FUNCTION_BLOCK CRANE_1_PUBLISH (* Composite Function Block Type *)
  (* Standard: 61499-2 *)
  (* Version 1.0, 2019-04-13, adeel *)
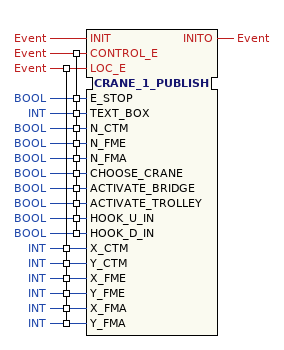
  EVENT_INPUT
    INIT; (* Initialization Request *)
    CONTROL_E WITH E_STOP, TEXT_BOX, N_CTM, N_FME, N_FMA, CHOOSE_CRANE, ACTIVATE_BRIDGE, ACTIVATE_TROLLEY, HOOK_U_IN, HOOK_D_IN; (* Normal Execution Request *)
    LOC_E WITH X_CTM, Y_CTM, X_FME, Y_FME, X_FMA, Y_FMA;
  END_EVENT
  EVENT_OUTPUT
    INITO; (* Initialization Confirm *)
  END_EVENT
  VAR_INPUT
    E_STOP : BOOL;
    TEXT_BOX : INT;
    N_CTM : BOOL;
    N_FME : BOOL;
    N_FMA : BOOL;
    CHOOSE_CRANE : BOOL;
    ACTIVATE_BRIDGE : BOOL;
    ACTIVATE_TROLLEY : BOOL;
    HOOK_U_IN : BOOL;
    HOOK_D_IN : BOOL;
    X_CTM : INT;
    Y_CTM : INT;
    X_FME : INT;
    Y_FME : INT;
    X_FMA : INT;
    Y_FMA : INT;
  END_VAR
  FBS
    PUBLISH_1 : PUBLISH_1(QI := 1, ID := opc_ua[opc.tcp://%CRANE1_IP%:4840#/Objects/1:CRANE1C/N_CTM/IN]);
    PUBLISH_1_1 : PUBLISH_1(QI := 1, ID := opc_ua[opc.tcp://%CRANE1_IP%:4840#/Objects/1:CRANE1B/TEXT_BOX/IN]);
    PUBLISH_1_2 : PUBLISH_1(QI := 1, ID := opc_ua[opc.tcp://%CRANE1_IP%:4840#/Objects/1:CRANE1K/X_CTM/IN]);
    PUBLISH_1_3 : PUBLISH_1(QI := 1, ID := opc_ua[opc.tcp://%CRANE1_IP%:4840#/Objects/1:CRANE1A/E_STOP/IN]);
    PUBLISH_1_4 : PUBLISH_1(QI := 1, ID := opc_ua[opc.tcp://%CRANE1_IP%:4840#/Objects/1:CRANE1L/Y_CTM/IN]);
    PUBLISH_1_5 : PUBLISH_1(QI := 1, ID := opc_ua[opc.tcp://%CRANE1_IP%:4840#/Objects/1D:CRANE1/N_FME/IN]);
    PUBLISH_1_6 : PUBLISH_1(QI := 1, ID := opc_ua[opc.tcp://%CRANE1_IP%:4840#/Objects/1:CRANE1O/X_FMA/IN]);
    PUBLISH_1_7 : PUBLISH_1(QI := 1, ID := opc_ua[opc.tcp://%CRANE1_IP%:4840#/Objects/1:CRANE1P/Y_FMA/IN]);
    PUBLISH_1_8 : PUBLISH_1(QI := 1, ID := opc_ua[opc.tcp://%CRANE1_IP%:4840#/Objects/1:CRANE1F/CHOOSE_CRANE/IN]);
    PUBLISH_1_9 : PUBLISH_1(QI := 1, ID := opc_ua[opc.tcp://%CRANE1_IP%:4840#/Objects/1:CRANE1H/ACTIVATE_TROLLEY/IN]);
    PUBLISH_1_10 : PUBLISH_1(QI := 1, ID := opc_ua[opc.tcp://%CRANE1_IP%:4840#/Objects/1:CRANE1I/HOOK_U_IN/IN]);
    PUBLISH_1_11 : PUBLISH_1(QI := 1, ID := opc_ua[opc.tcp://%CRANE1_IP%:4840#/Objects/1:CRANE1H/ACTIVATE_BRIDGE/IN]);
    PUBLISH_1_12 : PUBLISH_1(QI := 1, ID := opc_ua[opc.tcp://%CRANE1_IP%:4840#/Objects/1:CRANE1E/N_FMA/IN]);
    PUBLISH_1_13 : PUBLISH_1(QI := 1, ID := opc_ua[opc.tcp://%CRANE1_IP%:4840#/Objects/1:CRANE1J/HOOK_D_IN/IN]);
    PUBLISH_1_14 : PUBLISH_1(QI := 1, ID := opc_ua[opc.tcp://%CRANE1_IP%:4840#/Objects/1:CRANE1M/X_FME/IN]);
    PUBLISH_1_15 : PUBLISH_1(QI := 1, ID := opc_ua[opc.tcp://%CRANE1_IP%:4840#/Objects/1:CRANE1N/Y_FME/IN]);
  END_FBS
  EVENT_CONNECTIONS
    LOC_E TO PUBLISH_1_2.REQ;
    INIT TO PUBLISH_1_3.INIT;
    PUBLISH_1_3.INITO TO PUBLISH_1_1.INIT;
    PUBLISH_1_1.INITO TO PUBLISH_1.INIT;
    PUBLISH_1.INITO TO PUBLISH_1_5.INIT;
    PUBLISH_1_5.INITO TO PUBLISH_1_12.INIT;
    PUBLISH_1_12.INITO TO PUBLISH_1_8.INIT;
    PUBLISH_1_8.INITO TO PUBLISH_1_11.INIT;
    PUBLISH_1_11.INITO TO PUBLISH_1_9.INIT;
    PUBLISH_1_9.INITO TO PUBLISH_1_10.INIT;
    PUBLISH_1_10.INITO TO PUBLISH_1_13.INIT;
    PUBLISH_1_13.INITO TO PUBLISH_1_2.INIT;
    PUBLISH_1_2.INITO TO PUBLISH_1_4.INIT;
    PUBLISH_1_4.INITO TO PUBLISH_1_14.INIT;
    PUBLISH_1_14.INITO TO PUBLISH_1_15.INIT;
    PUBLISH_1_15.INITO TO PUBLISH_1_6.INIT;
    PUBLISH_1_6.INITO TO PUBLISH_1_7.INIT;
    PUBLISH_1_7.INITO TO INITO;
    LOC_E TO PUBLISH_1_4.REQ;
    LOC_E TO PUBLISH_1_14.REQ;
    LOC_E TO PUBLISH_1_15.REQ;
    LOC_E TO PUBLISH_1_6.REQ;
    LOC_E TO PUBLISH_1_7.REQ;
    CONTROL_E TO PUBLISH_1_3.REQ;
    CONTROL_E TO PUBLISH_1_1.REQ;
    CONTROL_E TO PUBLISH_1.REQ;
    CONTROL_E TO PUBLISH_1_5.REQ;
    CONTROL_E TO PUBLISH_1_12.REQ;
    CONTROL_E TO PUBLISH_1_8.REQ;
    CONTROL_E TO PUBLISH_1_11.REQ;
    CONTROL_E TO PUBLISH_1_9.REQ;
    CONTROL_E TO PUBLISH_1_10.REQ;
    CONTROL_E TO PUBLISH_1_13.REQ;
  END_CONNECTIONS
  DATA_CONNECTIONS
    X_CTM TO PUBLISH_1_2.SD_1;
    Y_CTM TO PUBLISH_1_4.SD_1;
    X_FME TO PUBLISH_1_14.SD_1;
    Y_FME TO PUBLISH_1_15.SD_1;
    X_FMA TO PUBLISH_1_6.SD_1;
    Y_FMA TO PUBLISH_1_7.SD_1;
    E_STOP TO PUBLISH_1_3.SD_1;
    TEXT_BOX TO PUBLISH_1_1.SD_1;
    N_CTM TO PUBLISH_1.SD_1;
    N_FME TO PUBLISH_1_5.SD_1;
    N_FMA TO PUBLISH_1_12.SD_1;
    CHOOSE_CRANE TO PUBLISH_1_8.SD_1;
    ACTIVATE_BRIDGE TO PUBLISH_1_11.SD_1;
    ACTIVATE_TROLLEY TO PUBLISH_1_9.SD_1;
    HOOK_U_IN TO PUBLISH_1_10.SD_1;
    HOOK_D_IN TO PUBLISH_1_13.SD_1;
  END_CONNECTIONS
END_FUNCTION_BLOCK
